PROGRAM MAIN
VAR
	fbAlarmCore : FB_AlarmCore;
	fbAlarm		: FB_Alarm;
	
	addAlarm	: BOOL;
END_VAR

IF addAlarm THEN
	fbAlarm.RaiseAlarm('This is Info from main program');
	addAlarm := FALSE;
END_IF

SecondUnit();

END_PROGRAM

(* stored: Version 1.1.0.1, ProductVersion 3.1.4026.6
   POU MAIN: Id {5ea28249-cb4a-49a2-996f-28f51da6431f}, SpecialFunc None *)
